{attribute 'qualified_only'}
VAR_GLOBAL CONSTANT
    // ── Valve motion parameters ───────────────────────────────
    VALVE_FULL_STROKE_MM           : REAL  := 6.096;     // Mechanical full travel for 0..100% scaling
    VALVE_POSITION_TOLERANCE       : REAL  := 0.5;       // In-position dead-band in percent
    VALVE_MOVE_VELOCITY            : LREAL := 1.5;       // mm/s
    VALVE_MOVE_ACCELERATION        : LREAL := 16.9085;   // mm/s²
    VALVE_MOVE_DECELERATION        : LREAL := 16.9085;   // mm/s²
    VALVE_MOVE_JERK                : LREAL := 53.5391;   // mm/s³
    VALVE_HOMING_VELOCITY          : LREAL := 1.0;       // Reference only (NC axis settings still apply)

    // ── CSV Logging ───────────────────────────────────────────
    CSV_LOG_INTERVAL_S             : TIME   := T#15M;
    CSV_FILE_PATH                  : STRING := 'C:\TwinCAT\3.1\Boot\Log\';
    CSV_FILENAME_PREFIX            : STRING := 'IrrigationLog_';

    // ── MQTT defaults (single source of truth) ───────────────
    // These are copied into ST_MqttConfig in MAIN on startup.
    // HMI only controls enable/disable, not broker parameter editing.
    MQTT_DEFAULT_BROKER_IP         : STRING := '192.168.1.100';
    MQTT_DEFAULT_PORT              : UINT   := 1883;
    MQTT_DEFAULT_CLIENT_ID         : STRING := 'BeckhoffIrrigationPLC';
    MQTT_DEFAULT_USERNAME          : STRING := '';
    MQTT_DEFAULT_PASSWORD          : STRING := '';
    MQTT_DEFAULT_USE_TLS           : BOOL   := FALSE;

    MQTT_DEFAULT_TOPIC_PREFIX      : STRING := 'irrigation';
    MQTT_STATUS_TOPIC              : STRING := 'irrigation/status';
    MQTT_COMMAND_TOPIC             : STRING := 'irrigation/command';

    MQTT_PUBLISH_INTERVAL          : TIME   := T#5M;
    MQTT_RECONNECT_DELAY           : TIME   := T#30S;

    // ── Task cycle time ───────────────────────────────────────
    TASK_CYCLE_MS                  : UINT := 10;         // Must match TwinCAT task setting
END_VAR

(* stored: Version 1.1.0.1, ProductVersion 3.1.4026.18
   GVL GVL_Config: Id {3f9b61cc-9b72-4973-88f0-22ca8b080aec} *)
